FUNCTION_BLOCK FB_Simple
VAR_INPUT
    rSollwert  : REAL;
    rIstwert   : REAL;
    bAktiv     : BOOL;
END_VAR
VAR_OUTPUT
    rStellwert : REAL;
    bFehler    : BOOL;
END_VAR
VAR
    rFehler    : REAL;
    rIntegral  : REAL;
    rKp        : REAL := 1.0;
    rKi        : REAL := 0.1;
END_VAR
VAR_TEMP
    rTemp      : REAL;
END_VAR

BEGIN
    IF bAktiv THEN
        rFehler   := rSollwert - rIstwert;
        rIntegral := rIntegral + rFehler * rKi;
        rTemp     := rKp * rFehler + rIntegral;
        rStellwert := rTemp;
        bFehler    := FALSE;
    ELSE
        rStellwert := 0.0;
        bFehler    := TRUE;
    END_IF;
END_FUNCTION_BLOCK
